// TIA Portal V17 export
// export: Created 2024-01-30T08:49:13.2459545Z, ExportSetting WithDefaults, DisplayName Totally Integrated Automation Portal, DisplayVersion V17 Update 6, DisplayName TIA Portal Openness, DisplayVersion V17 Update 6, DisplayName TIA Portal Version Control Interface, DisplayVersion V17, DisplayName STEP 7 Professional, DisplayVersion V17 Update 6, DisplayName STEP 7 Safety, DisplayVersion V17 Update 6, DisplayName WinCC Advanced, DisplayVersion V17 Update 6
DATA_BLOCK "GDB_LJ_X8000"   // DB10
{ S7_Optimized_Access := 'TRUE' }
VERSION : 0.1
// stored: AutoNumber true, DBAccessibleFromOPCUA true, DBAccessibleFromWebserver true, IsOnlyStoredInLoadMemory false, IsRetainMemResEnabled false, IsWriteProtectedInAS false, MemoryReserve 100
   VAR
      PLC_to_LJX8000bits : "UDT_PLC --> LJ_X8000_Bits";
      PLC_to_LJX8000bytes { S7_SetPoint := 'True'} : "UDT_PLC --> LJ_X8000_Bytes";
      LJX8000_to_PLCbits { S7_SetPoint := 'True'} : "UDT_LJ_X8000 --> PLC_Bits";
      LJX8000_to_PLCbytes { S7_SetPoint := 'True'} : "UDT_LJ_X8000 --> PLC_Bytes";
      CTRL : Struct
         UserCommand : Int;
         ProgramNumber : Int;
         ResetError : Bool;
         CommandRequest : Bool;
         Trigger : Bool;
      END_STRUCT;
      HMI : Struct
         StartMeasurement : Bool;
         MeasurementMode : Bool;
         HandMode : Bool;
         CellType : SInt;
         SQ_ActivTask : SInt;
      END_STRUCT;
      Cell_MeasData : Struct
         Länge : Real;
         Breite : Real;
      END_STRUCT;
   END_VAR
BEGIN
END_DATA_BLOCK
